FUNCTION AddREAL : BOOL				// Increments the given UINT value
VAR_INPUT
	iAdd:	REAL;
END_VAR
VAR_IN_OUT
	ioNum:	REAL;		// Value to increment
END_VAR

ioNum := ioNum + iAdd;

END_FUNCTION

(* stored: Version 1.1.0.1, ProductVersion 3.1.4026.18
   POU AddREAL: Id {89cc04ef-ba49-4788-8c60-99b1c3e34711}, SpecialFunc None *)
